FUNCTION CallHardwareModules : BOOL //only purpose of this function is to call modules from Hardware
VAR_STAT
	temp : INT;
END_VAR

robot1();	
robot2();

//(*
temp := TO_INT(BoolArrayToInteger(arr := stagingTableLeft.occupied));
temp.15 := NOT strapperA21.bEnable AND NOT strapperA21.execute;
robot1.setGroup(group := 8, value := temp);

temp := TO_INT(BoolArrayToInteger(arr := stagingTableRight.occupied));
temp.15 := NOT strapperA21.bEnable AND NOT strapperA21.execute;
robot2.setGroup(group := 8, value := temp);
//*)

skidA21Left();
skidA21Right();

stagingTableLeft();
stagingTableRight();

skidA21Left();
skidA21Right();

magazineA21Left();
magazineA21Right();

stagingTableLeft();
stagingTableRight();

strapperA21();

verticalDriveA21Left();
verticalDriveA21Right();
horizontalDriveA21Left();
horizontalDriveA21Right();
pistonA21Bottom();

END_FUNCTION

(* stored: Version 1.1.0.1, ProductVersion 3.1.4024.11
   POU CallHardwareModules: Id {d53bfde7-ef31-4033-a59e-17a8585cdf25}, SpecialFunc None *)
